{attribute addProperty BoxType "EJ7031-0000-0026"}
{attribute addProperty Id "AdsAddrAT %I*AMSADDR6480Chn0AT %I*USINT810Chn1AT %I*USINT810StateAT %I*UINT1620"}
{attribute addProperty CRC "474407911"}
{attribute addProperty SizeInBites "96"}
{attribute addProperty SizeInBytes "12"}
TYPE InfoData_1C46E3E7 :
STRUCT
	{attribute addProperty Name "AdsAddr"}
	AdsAddr AT %I* : AMSADDR;
	{attribute addProperty Name "Chn0"}
	Chn0 AT %I* : USINT;
	{attribute addProperty Name "Chn1"}
	Chn1 AT %I* : USINT;
	{attribute addProperty Name "State"}
	State AT %I* : UINT;
END_STRUCT
END_TYPE

(* stored: Version 1.2.0.0, ProductVersion 3.1.4024.9
   DUT InfoData_1C46E3E7: Id {6982bc09-4fae-4e45-bac3-9af49e618cf6} *)
